// TIA Portal project "First" (V17)

(* hardware
DEVICE "S7-1200 station_1"  S7-1200 Station
   slot 0: "Rack_0"  S7-1200 Rack  Rack  V1.0
   slot 1: "SIMATIC_S7_1214C"  CPU 1214C DC/DC/DC  6ES7 214-1AG31-0XB0  V3.0
   slot 101: "CM 1241 (RS485)_1"  CM 1241 (RS485)  6ES7 241-1CH30-0XB0  V1.0
DEVICE "S7-1200 station_2"  S7-1200 Station
   slot 0: "Rack_0"  S7-1200 Rack  Rack  V1.0
   slot 1: "PLC_1"  CPU 1214C DC/DC/DC  6ES7 214-1AG40-0XB0  V4.5
*)

// ===== PLC "SIMATIC_S7_1214C"  CPU 1214C DC/DC/DC =====

VAR_GLOBAL   // PLC tag table "Default tag table"
   "DO01" AT %Q0.0 : Bool;
   "DI01" AT %I0.0 : Bool;
   "DO02" AT %Q0.1 : Bool;
   "DO04" AT %Q0.2 : Bool;
END_VAR

DATA_BLOCK "Data_block_1"   // DB4
{ S7_Optimized_Access := 'TRUE' }
VERSION : 0.1
   VAR
      "M0.1" : Bool;
   END_VAR
BEGIN
END_DATA_BLOCK

// folder: System blocks/Program resources

DATA_BLOCK "IEC_Timer_0_DB"   // DB1
{ S7_Optimized_Access := 'TRUE' }
AUTHOR : Simatic
FAMILY : IEC
NAME : IEC_TMR
VERSION : 1.0
// stored: InstanceOfName IEC_TIMER
"IEC_TIMER"
BEGIN
END_DATA_BLOCK

DATA_BLOCK "IEC_Timer_0_DB_1"   // DB3
{ S7_Optimized_Access := 'TRUE' }
AUTHOR : Simatic
FAMILY : IEC
NAME : IEC_TMR
VERSION : 1.0
// stored: InstanceOfName IEC_TIMER
"IEC_TIMER"
BEGIN
END_DATA_BLOCK

DATA_BLOCK "IEC_Timer_0_DB_2"   // DB5
{ S7_Optimized_Access := 'TRUE' }
AUTHOR : Simatic
FAMILY : IEC
NAME : IEC_TMR
VERSION : 1.0
// stored: InstanceOfName IEC_TIMER
"IEC_TIMER"
BEGIN
END_DATA_BLOCK

DATA_BLOCK "IEC_Timer_0_DB_3"   // DB6
{ S7_Optimized_Access := 'TRUE' }
AUTHOR : Simatic
FAMILY : IEC
NAME : IEC_TMR
VERSION : 1.0
// stored: InstanceOfName IEC_TIMER
"IEC_TIMER"
BEGIN
END_DATA_BLOCK

DATA_BLOCK "IEC_Timer_0_DB_4"   // DB7
{ S7_Optimized_Access := 'TRUE' }
AUTHOR : Simatic
FAMILY : IEC
NAME : IEC_TMR
VERSION : 1.0
// stored: InstanceOfName IEC_TIMER
"IEC_TIMER"
BEGIN
END_DATA_BLOCK

DATA_BLOCK "IEC_Timer_0_DB_5"   // DB8
{ S7_Optimized_Access := 'TRUE' }
AUTHOR : Simatic
FAMILY : IEC
NAME : IEC_TMR
VERSION : 1.0
// stored: InstanceOfName IEC_TIMER
"IEC_TIMER"
BEGIN
END_DATA_BLOCK

// folder: (top level)

ORGANIZATION_BLOCK "Main"   // OB1, LAD, ProgramCycle
TITLE = "Main Program Sweep (Cycle)"
{ S7_Optimized_Access := 'TRUE' }
VERSION : 0.1
BEGIN

REGION Network 1
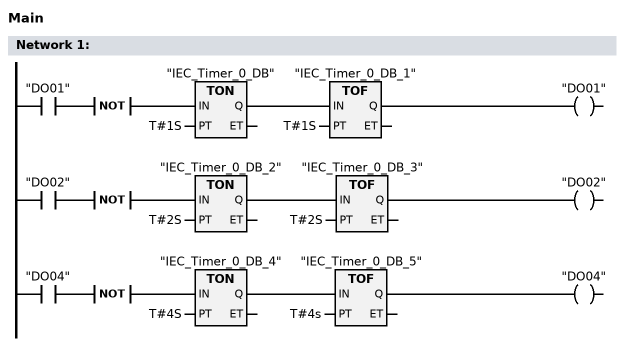
   "IEC_Timer_0_DB".TON(IN := NOT "DO01", PT := T#1S);
   "IEC_Timer_0_DB_1".TOF(IN := "IEC_Timer_0_DB".Q, PT := T#1S);
   "DO01" := "IEC_Timer_0_DB_1".Q;
   "IEC_Timer_0_DB_2".TON(IN := NOT "DO02", PT := T#2S);
   "IEC_Timer_0_DB_3".TOF(IN := "IEC_Timer_0_DB_2".Q, PT := T#2S);
   "DO02" := "IEC_Timer_0_DB_3".Q;
   "IEC_Timer_0_DB_4".TON(IN := NOT "DO04", PT := T#4S);
   "IEC_Timer_0_DB_5".TOF(IN := "IEC_Timer_0_DB_4".Q, PT := T#4s);
   "DO04" := "IEC_Timer_0_DB_5".Q;
END_REGION
END_ORGANIZATION_BLOCK

// folder: LGF/7 Signal generators

FUNCTION_BLOCK "LGF_RectangleCI"   // FB10029, SCL
TITLE = LGF_RectangleCI
{ S7_Optimized_Access := 'TRUE' }
AUTHOR : Siemens_Industry_Support
FAMILY : LGF
NAME : LGF_RectangleCI
// This function generates a rectangular signal profile. For this it uses the time interval of the calling Cyclic Interrupt OB. / Diese Funktion generiert einen rechteckigen Signalverlauf. Er verwendet dazu den Zeittakt des aufrufenden Cyclic Interrupt OB.
   VAR_INPUT
      amplitude : Real := 1.0;   // Amplitude of the signal profile. / Amplitude des Signalverlaufs.
      offset : Real;   // Offset of the signal profile in the Y-direction. / Verschiebung des Signalverlaufs in Y-Richtung.
      periode : UDInt := 1000;   // Period duration of the signal profile in [ms] / Periodendauer des Signalverlaufs in [ms]
      phaseShift : Real;   // Phase offset in [ms] / Phasenverschiebung in [ms]
      callOB : OB_Cyclic;   // Calling cyclic interrupt OB / Aufrufender Weckalarm-OB (Cyclic Interrupt OB)
      reset : Bool;   // Reset of the signal profile. / Rücksetzen des Signalverlaufs.
   END_VAR
   VAR_OUTPUT
      value : Real;   // Current value of the rectangular signal. / Aktueller Wert des Rechtecksignales.
      error : Bool;   // FALSE: No error TRUE: An error occurred during the execution of the FB / FALSE: Kein Fehler TRUE: Während der Ausführung des FB ist ein Fehler aufgetreten
      status : Word := 16#0;   // 16#0000-16#7FFF: Status of the FB 16#8000-16#FFFF: Error identification (see following Table) / 16#0000-16#7FFF: Status des FB 16#8000-16#FFFF: Fehleridentifikation (siehe folgende Tabelle)
      subFunctionStatus : Word := 16#0;   // Status or return value of called FB's, FC's and system blocks / Status oder Rückgabewert von aufgerufenen FB's / FC's und Systemfunktionen
   END_VAR
   VAR
      statCounter : UDInt;   // Static Counter value
   END_VAR
   VAR_TEMP
      tempCycleTime : UDInt;   // Temp cycle time from CallOB
      tempCyclePhase : UDInt;   // Temp cycle phase from CallOB
      tempCycleStatus : Word;   // Temp cycle status from CallOB
      tempReadTimeStatus : Int;   // Temp return value of QRY_CINT
      tempValue : Real;   // Temp output value
      tempPhaseShift : UDInt;   // Temp phase shift value MODULO periode
   END_VAR
   VAR CONSTANT
      SECOND_IN_MS : UDInt := 1000;   // One second written in milliseconds. Needed in calculation in formulas / One second written in miliseconds. Needed in calculation in formulas
      ZERO : Int := 0;   // Numeric zero value
      RATIO : UDInt := 2;   // Ratio = used to calculate the half period
      SUB_STATUS_NO_ERROR : Word := 16#0000;   // Subfunction status: No error
      STATUS_FINISHED_NO_ERROR : Word := 16#0000;   // Status: Execution finished without errors / Status: Abarbeitung ohne Fehler beendet
      QRY_CINT_OB_UNAVAILABLE : Word := 16#0000;   // Cyclic interrupt status: OB not available
      ERR_OB_UNAVAILABLE : Word := 16#8600;   // Error: OB on input `callOB` is not configured / present. Interconnect the constant name of a configured cyclic interrupt OB at the input `callOB`. / Fehler: OB am Eingang `callOB` ist nicht projektiert / vorhanden. Verschalten Sie am Eingang `callOB` den Konstanten Namen eines projektierten Weckalarm-OB.
      ERR_QRY_CINT : Word := 16#8601;   // Error in `QRY_CINT` command - check `subFunctionStatus` code / Fehler in Anweisung `QRY_CINT` - weitere Infos in `subFunctionStatus`
   END_VAR
BEGIN
   REGION Block info header
     //===============================================================================
     // SIEMENS AG / (c)Copyright 2019
     //-------------------------------------------------------------------------------
     // Title:            LGF_RectangleCI
     // Comment/Function: This function generates a rectangular signal profile. For this it uses the time interval of the calling Cyclic Interrupt OB.
     // Library/Family:   LGF (Library General Functions)
     // Author:           Siemens Digital Industry Support
     // Tested with:      CPU 1515F-2 PN FW:V2.6
     // Engineering:      TIA Portal V15.1 Update 2
     // Restrictions:     ENO disabled - error handling done by error and status
     // Requirements:     PLC (S7-1200 / S7-1500)
     //-------------------------------------------------------------------------------
     // Change log table:
     // Version  | Date       | Expert in charge       | Changes applied
     //----------|------------|------------------------|------------------------------
     // 01.00.00 03.07.2018  Siemens Industry Online Support
     //                      First released version
     // 01.00.01 17.08.2018  Siemens Industry Online Support
     //                      Upgrade: TIA V15 Update 2
     // 01.00.02 23.11.2018  Siemens Industry Online Support
     //                      Upgrade: TIA V15.1
     // 01.00.03 26.09.2019  Simatic Systems Support
     //                      Code refactoring, regions and more comments added
     //                      phase shift availability added
     // 03.00.00 23.04.2020  Simatic Systems Support
     //                      Set version to V3.0.0, harmonize the version of the whole library
     // 03.00.01 15.02.2021  Simatic Systems Support
     //                      Insert documentation
     //=============================================================================
   END_REGION Block info header

   REGION DESCRIPTION
     (/*NOTE
   :    The status of called commands is output in `subFunctionStatus`. In this case, the output value in `status` indicates which command caused the error. In this case, refer to the TIA Portal Online Help section for information on the respective commands.

   ---

   The block calculates the values for a rectangular signal profile, which is output to the output parameter `value`.

   The `amplitude`, the `offset` in the Y-direction, the `period`, and the `phase shift` can be set at the input parameters.

   The input parameter `reset` resets the signal profile. At the `value` output parameter, the value `0` is output as long as `reset` is set to `TRUE`.

   The block must be called in a cyclic interrupt OB. The time interval of the calling cyclic interrupt OB is determined in the FB with the command `QRY_CINT`. For this, the constant name of the calling cyclic interrupt OB must be interconnected at the input parameter `callOB`.

   ![Interconnecting the cyclic interrupt OB](LGF_InterruptObAsParameter.png "Interconnecting the cyclic interrupt OB")

   The number of calculated values of the signal profile per period duration is calculated as follows:

   $$
     Quantity Values = \frac{Period duration}{Time intervak Cyclic interrupt OB}
   $$

   ---

   Note
   :    To obtain a continuous signal profile of the curve, the time interval of the cyclic interrupt OB should not be selected too large depending on the period duration.

   ---

   ------

   The Figure below shows the signal profile of the calculated values.

   ![LGF_RectangleCI](LGF_RectangleCI.png "LGF_RectangleCI")
   Hinweis
   :    In `subFunctionStatus` wird der Status von aufgerufenen Anweisungen ausgegeben. Der Ausgangswert in `status` gibt in diesem Fall an, welche Anweisung den Fehler verursacht hat. Holen Sie sich in diesem Fall die Informationen aus der TIA Portal Online Hilfe zu den jeweiligen Anweisungen.

   ---

   Der Baustein berechnet die Werte für einen rechteckigen Signalverlauf, die am Ausgangsparameter `value` ausgegeben werden.

   Die Amplitude `amplitude`, die Verschiebung in Y-Richtung `offset`, die Periodendauer `periode` und die Phasenverschiebung `phaseShift` können an den Eingangsparametern vorgegeben werden.

   Mit dem Eingangsparameter `reset` wird der Signalverlauf zurückgesetzt. Am Ausgangsparameter `value` wird der Wert `0` ausgegeben, solange `reset` auf `TRUE` gesetzt ist.

   Der Baustein muss in einem Weckalarm-OB (Cyclic Interrupt OB) aufgerufen werden. Der Zeittakt des aufrufenden Weckalarm-OB wird im FB mit der Anweisung `QRY_CINT` ermittelt. Dazu muss am Eingangsparameter `callOB` der Konstanten Name des aufrufenden Weckalarm-OB verschaltet werden.

   ![Weckalarm-OB verschalten](LGF_InterruptObAsParameter.png "Weckalarm-OB verschalten")

   Die Anzahl der berechneten Werte des Signalverlaufs pro Periodendauer errechnet sich folgendermaßen:

   $$
     Anzahl Werte = \frac{Periodendauer}{Zeittakt Weckalarm-OB}
   $$

   ---

   Hinweis
   :    Um einen kontinuierlichen Signalverlauf der Kurve zu erhalten, sollte der Zeittakt des aufrufen Weckalarm-OB in Abhängigkeit von der Periodendauer nicht zu groß gewählt werden.

   ---

   ------

   Die folgende Abbildung zeigt den Signalverlauf der berechneten Werte.

   ![LGF_RectangleCI](LGF_RectangleCI.png "LGF_RectangleCI")*/)
   END_REGION DESCRIPTION

   REGION Get sample time
     // get sample time, according to the cyclic interrupt OB number
     #tempReadTimeStatus := QRY_CINT(OB_NR := #callOB, CYCLE => #tempCycleTime,
                                     PHASE => #tempCyclePhase, STATUS => #tempCycleStatus);

     REGION Error handling
       // Generate error message of the QRY_CINT function
       IF #tempReadTimeStatus <> #ZERO THEN
         #error := TRUE;
         #status := #ERR_QRY_CINT;
         #subFunctionStatus := INT_TO_WORD(#tempReadTimeStatus);
         #value := #ZERO;
         RETURN;

         // Generate error message when OB unavailable
       ELSIF (#tempCycleStatus = #QRY_CINT_OB_UNAVAILABLE) THEN
         #error := TRUE;
         #status := #ERR_OB_UNAVAILABLE;
         #subFunctionStatus := #SUB_STATUS_NO_ERROR;
         #value := #ZERO;
         RETURN;
       END_IF;
     END_REGION
   END_REGION

   REGION Caluclations and outputs assigment
     // calculate true phase shift with modulo
     #tempPhaseShift := REAL_TO_UDINT(#phaseShift) MOD #periode;

     IF #reset THEN
       #statCounter := #tempPhaseShift;
       #tempValue := #ZERO;
     ELSE
       // Increment Counter with each call of "OB_Cyclic_interrupt"
       #statCounter += #tempCycleTime / #SECOND_IN_MS;
       #statCounter := #statCounter MOD #periode;

       // Calculate output value
       #tempValue := #offset;

       IF (#statCounter >= #tempPhaseShift) AND (#statCounter < (#periode / #RATIO) + #tempPhaseShift) THEN
         #tempValue += #amplitude;
       ELSE
         #tempValue -= #amplitude;
       END_IF;
     END_IF;

     #value := #tempValue;
     #error := FALSE;
     #status := #STATUS_FINISHED_NO_ERROR;
     #subFunctionStatus := #SUB_STATUS_NO_ERROR;
     //ENO mechanism is not used - forced to true.
     ENO := TRUE;
   END_REGION
END_FUNCTION_BLOCK

// ===== PLC "PLC_1"  CPU 1214C DC/DC/DC =====

VAR_GLOBAL   // PLC tag table "Default tag table"
   "DO01" AT %Q0.0 : Bool;
END_VAR

// folder: System blocks/Program resources

DATA_BLOCK "IEC_Timer_0_DB_1"   // DB1
{ S7_Optimized_Access := 'TRUE' }
AUTHOR : Simatic
FAMILY : IEC
NAME : IEC_TMR
VERSION : 1.0
// stored: InstanceOfName IEC_TIMER
"IEC_TIMER"
BEGIN
END_DATA_BLOCK

DATA_BLOCK "IEC_Timer_0_DB_2"   // DB2
{ S7_Optimized_Access := 'TRUE' }
AUTHOR : Simatic
FAMILY : IEC
NAME : IEC_TMR
VERSION : 1.0
// stored: InstanceOfName IEC_TIMER
"IEC_TIMER"
BEGIN
END_DATA_BLOCK

// folder: (top level)

ORGANIZATION_BLOCK "Main"   // OB1, LAD, ProgramCycle
TITLE = "Main Program Sweep (Cycle)"
{ S7_Optimized_Access := 'TRUE' }
VERSION : 0.1
   VAR_INPUT
      Initial_Call : Bool;   // Initial call of this OB
      Remanence : Bool;   // =True, if remanent data are available
   END_VAR
BEGIN

REGION Network 1
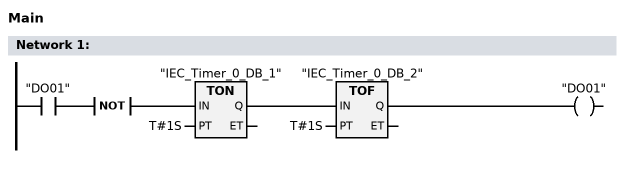
   "IEC_Timer_0_DB_1".TON(IN := NOT "DO01", PT := T#1S);
   "IEC_Timer_0_DB_2".TOF(IN := "IEC_Timer_0_DB_1".Q, PT := T#1S);
   "DO01" := "IEC_Timer_0_DB_2".Q;
END_REGION
END_ORGANIZATION_BLOCK